KUKA KRL data list: tipdress1.dat

&ACCESS RV1
&REL 49
&COMMENT TIPDRESS EXTERNAL GUN 1
DEFDAT  TIPDRESS1
;FOLD EXTERNAL DECLARATIONS;%{PE}%MKUKATPBASIS,%CEXT,%VCOMMON,%P
;FOLD GRIPPERTECH EXT
EXT  H50 (INT  :IN,INT  :IN,INT  :IN,GRP_TYP  :IN )
;ENDFOLD (GRIPPERTECH EXT)
;FOLD SPOTTECH EXT
EXT  USERSPOT (S_COMMAND  :IN,SPOT_TYPE  :IN )
;ENDFOLD (SPOTTECH EXT)
;FOLD BASISTECH EXT;%{PE}%MKUKATPBASIS,%CEXT,%VEXT,%P
EXT  BAS (BAS_COMMAND  :IN,REAL  :IN )
DECL INT SUCCESS
;ENDFOLD (BASISTECH EXT)
;FOLD USER EXT;%{E}%MKUKATPUSER,%CEXT,%VEXT,%P
;Make here your modifications
;ENDFOLD (USER EXT)
;ENDFOLD (EXTERNAL DECLERATIONS)
;FOLD USER EXT;%{}%V2.2.2,%MKUKATPUSER,%CEXT,%VEXT,%P
;Make here your modifications
DECL BOOL TIPKONTROLE
DECL INT ANSWER
DECL INT WAITTIME=5
;ENDFOLD
;ENDFOLD
DECL INT I

;******************************
;*     E6POS Declarations     *
;******************************

DECL E6POS XP10={X 30.7658501,Y -1094.01099,Z -286.682404,A 25.4987392,B 1.97903597,C -0.329104304,S 6,T 26,E1 0.0,E2 0.0,E3 0.0,E4 0.0,E5 0.0,E6 0.0}
DECL E6POS XP20={X -1662.00305,Y -1200.49304,Z 238.679993,A 92.3594437,B 77.6989288,C -175.853195,S 6,T 26,E1 -667.745789,E2 0.0,E3 0.0,E4 0.0,E5 0.0,E6 0.0}
DECL E6POS XBEFORETIPDRESS={X -1664.84497,Y -1195.28101,Z 131.821106,A 92.7083206,B 79.2879791,C -177.241806,S 6,T 26,E1 -667.74939,E2 0.0,E3 0.0,E4 0.0,E5 0.0,E6 0.0}
DECL E6POS XDRESS_POS={X -1664.83301,Y -1250.33301,Z 131.817993,A 92.7068863,B 79.2882233,C -177.243393,S 6,T 26,E1 -667.74762,E2 0.0,E3 0.0,E4 0.0,E5 0.0,E6 0.0}
DECL E6POS XAFTERTIPDRESS={X -1664.84497,Y -1195.28101,Z 131.821106,A 92.7083206,B 79.2879791,C -177.241806,S 6,T 26,E1 -667.74939,E2 0.0,E3 0.0,E4 0.0,E5 0.0,E6 0.0}
DECL E6POS XBEST_PRACKTICE={X -1662.02905,Y -1184.83496,Z 277.771301,A 92.3578873,B 77.6946869,C -175.853302,S 6,T 26,E1 -667.74762,E2 0.0,E3 0.0,E4 0.0,E5 0.0,E6 0.0}
DECL E6POS XP30={X -958.122009,Y 929.273499,Z 985.610474,A 92.0788727,B 72.5539932,C -179.8358,S 6,T 26,E1 -2887.17505,E2 0.0,E3 0.0,E4 0.0,E5 0.0,E6 0.0}

;******************************
;*      FDAT Declarations     *
;******************************

DECL FDAT FP10={TOOL_NO 1,BASE_NO 0,IPO_FRAME #BASE,TQ_STATE FALSE}
DECL FDAT FP20={TOOL_NO 1,BASE_NO 0,IPO_FRAME #BASE}
DECL FDAT FBEFORETIPDRESS={TOOL_NO 1,BASE_NO 0,IPO_FRAME #BASE}
DECL FDAT FDRESS_POS={TOOL_NO 1,BASE_NO 0,IPO_FRAME #BASE}
DECL FDAT FAFTERTIPDRESS={TOOL_NO 1,BASE_NO 0,IPO_FRAME #BASE}
DECL FDAT FBEST_PRACKTICE={TOOL_NO 1,BASE_NO 0,IPO_FRAME #BASE}
DECL FDAT FP30={TOOL_NO 1,BASE_NO 0,IPO_FRAME #BASE}

;******************************
;*  PDAT & LDAT Declarations  *
;******************************

DECL PDAT PH={VEL 100.0,ACC 100.0,APO_DIST 100.0,APO_MODE #CPTP}

DECL E6POS XBEST_PRAKTISCH={X 3.06066203,Y -1202.17297,Z 611.93042,A -125.567596,B -7.38407087,C -173.644897,S 6,T 26,E1 0.0,E2 0.0,E3 0.0,E4 0.0,E5 0.0,E6 0.0}
DECL SPOT_SUGG_T LAST_SPOT={GUN[] "1                       ",RETR_CMD[] "#OPN                    ",CHOISE[] "#FIRST                  ",CLO_TM[] "0                       ",PGNO1[] "1                       ",PRESS1[] "0                       ",PGNO2[] "1                       ",PRESS2[] "0                       ",SPOT_PARAMS[] "SDAT3                   "}
DECL BASIS_SUGG_T LAST_BASIS={POINT1[] "p1560                   ",POINT2[] "p1560                   ",CP_PARAMS[] "CPDAT0                  ",PTP_PARAMS[] "H                       ",CONT[] "C_PTP                   ",CP_VEL[] "2.0                     ",PTP_VEL[] "100                     ",SYNC_PARAMS[] "SYNCDAT                 ",SPL_NAME[] "S0                      "}
DECL FDAT FBest_Praktisch={TOOL_NO 14,BASE_NO 0,IPO_FRAME #BASE,POINT2[] " ",TQ_STATE FALSE}
DECL PDAT PPDAT1={VEL 100.0,ACC 100.0,APO_DIST 100.0}
DECL E6POS XBest_Praktice={X -1662.07202,Y -1184.76196,Z 277.795013,A 92.3631592,B 77.6921463,C -175.8461,S 6,T 26,E1 -667.74762,E2 0.0,E3 0.0,E4 0.0,E5 0.0,E6 0.0}
DECL FDAT FBest_Praktice={TOOL_NO 1,BASE_NO 0,IPO_FRAME #BASE,POINT2[] " "}
DECL E6POS XP21={X -929.55603,Y -159.533905,Z 748.283386,A 92.0804672,B 72.5703812,C -179.830597,S 6,T 26,E1 -2646.86792,E2 0.0,E3 0.0,E4 0.0,E5 0.0,E6 0.0}
DECL FDAT FP21={TOOL_NO 1,BASE_NO 0,IPO_FRAME #BASE}
DECL E6POS XP31={X -1185.09497,Y -662.41571,Z 415.422485,A 99.845192,B 75.8905869,C -168.599792,S 6,T 26,E1 -1294.38501,E2 0.0,E3 0.0,E4 0.0,E5 0.0,E6 0.0}
DECL FDAT FP31={TOOL_NO 1,BASE_NO 0,IPO_FRAME #BASE}
DECL E6POS XP01={X -521.268372,Y 932.237488,Z 809.362427,A -104.869499,B 25.3531094,C 156.8172,S 2,T 43,E1 0.0,E2 0.0,E3 0.0,E4 0.0,E5 0.0,E6 0.0}
DECL FDAT FP01={TOOL_NO 15,BASE_NO 0,IPO_FRAME #BASE,POINT2[] " ",TQ_STATE FALSE}
DECL E6POS XP02={X 1.47015905,Y -1176.46594,Z -326.900909,A 24.0927391,B 2.20976591,C -0.817254126,S 6,T 26,E1 0.0,E2 0.0,E3 0.0,E4 0.0,E5 0.0,E6 0.0}
DECL FDAT FP02={TOOL_NO 1,BASE_NO 0,IPO_FRAME #BASE,POINT2[] " ",TQ_STATE FALSE}
DECL E6POS XP022={X -545.304504,Y 780.863586,Z 303.431,A -96.6869965,B -0.146422103,C 179.108505,S 2,T 43,E1 0.0,E2 0.0,E3 0.0,E4 0.0,E5 0.0,E6 0.0}
DECL FDAT FP022={TOOL_NO 15,BASE_NO 0,IPO_FRAME #BASE,POINT2[] " ",TQ_STATE FALSE}
DECL E6POS XEXIT_FRESA={X -19.1423302,Y -1168.72705,Z 599.551025,A -125.410202,B 0.478198886,C -178.771393,S 6,T 26,E1 0.0,E2 0.0,E3 0.0,E4 0.0,E5 0.0,E6 0.0}
DECL FDAT Fexit_fresa={TOOL_NO 15,BASE_NO 0,IPO_FRAME #BASE,POINT2[] " ",TQ_STATE FALSE}
DECL E6POS XEXIT_FRESA_2={X -521.27002,Y 932.235901,Z 809.362793,A -104.869301,B 25.3530197,C 156.8172,S 2,T 43,E1 0.0,E2 0.0,E3 0.0,E4 0.0,E5 0.0,E6 0.0}
DECL FDAT Fexit_fresa_2={TOOL_NO 15,BASE_NO 0,IPO_FRAME #BASE,POINT2[] " ",TQ_STATE FALSE}
DECL E6POS XPRE_FRESADO={X 29.4938698,Y -1096.56396,Z -327.138885,A 25.4940891,B 1.89127803,C -0.142933503,S 6,T 26,E1 0.0,E2 0.0,E3 0.0,E4 0.0,E5 0.0,E6 0.0}
DECL FDAT Fpre_fresado={TOOL_NO 1,BASE_NO 0,IPO_FRAME #BASE,POINT2[] " ",TQ_STATE FALSE}
DECL E6POS XP1555={X 17.5958195,Y -1360.61597,Z -301.022308,A 23.6130409,B 6.36468601,C -9.25088882,S 6,T 26,E1 0.0,E2 0.0,E3 0.0,E4 0.0,E5 0.0,E6 0.0}
DECL FDAT Fp1555={TOOL_NO 1,BASE_NO 0,IPO_FRAME #BASE,POINT2[] " ",TQ_STATE FALSE}
DECL E6POS XP1556={X 481.643494,Y -1154.31702,Z -148.6595,A 30.6545601,B 3.87480402,C -9.08418941,S 6,T 26,E1 0.0,E2 0.0,E3 0.0,E4 0.0,E5 0.0,E6 0.0}
DECL FDAT Fp1556={TOOL_NO 1,BASE_NO 0,IPO_FRAME #BASE,POINT2[] " ",TQ_STATE FALSE}
DECL E6POS XP1557={X 735.259827,Y -846.376282,Z -50.7595787,A 36.4931488,B 2.33025098,C -7.71590185,S 6,T 26,E1 0.0,E2 0.0,E3 0.0,E4 0.0,E5 0.0,E6 0.0}
DECL FDAT Fp1557={TOOL_NO 1,BASE_NO 0,IPO_FRAME #BASE,POINT2[] " ",TQ_STATE FALSE}
DECL E6POS XP1558={X 415.015991,Y -1021.36499,Z 766.043091,A -118.665298,B -5.1592021,C -172.507797,S 6,T 26,E1 0.0,E2 0.0,E3 0.0,E4 0.0,E5 0.0,E6 0.0}
DECL FDAT Fp1558={TOOL_NO 15,BASE_NO 0,IPO_FRAME #BASE,POINT2[] " ",TQ_STATE FALSE}
DECL E6POS XP1559={X 648.731079,Y -753.047424,Z 867.173096,A -112.872597,B -3.13396502,C -172.896606,S 6,T 26,E1 0.0,E2 0.0,E3 0.0,E4 0.0,E5 0.0,E6 0.0}
DECL FDAT Fp1559={TOOL_NO 15,BASE_NO 0,IPO_FRAME #BASE,POINT2[] " ",TQ_STATE FALSE}
DECL E6POS XP1560={X 648.731079,Y -753.047424,Z 867.173096,A -112.872597,B -3.13396502,C -172.896606,S 6,T 26,E1 0.0,E2 0.0,E3 0.0,E4 0.0,E5 0.0,E6 0.0}
DECL FDAT Fp1560={TOOL_NO 15,BASE_NO 0,IPO_FRAME #BASE,POINT2[] " ",TQ_STATE FALSE}
DECL E6POS XP11={X 30.7658501,Y -1094.01099,Z -286.682404,A 25.4987392,B 1.97903597,C -0.329104304,S 6,T 26,E1 0.0,E2 0.0,E3 0.0,E4 0.0,E5 0.0,E6 0.0}
DECL FDAT FP11={TOOL_NO 1,BASE_NO 0,IPO_FRAME #BASE,TQ_STATE FALSE}
ENDDAT
